KUKA KRL program: sample_robot_pick_place.src, sample_robot_pick_place.dat

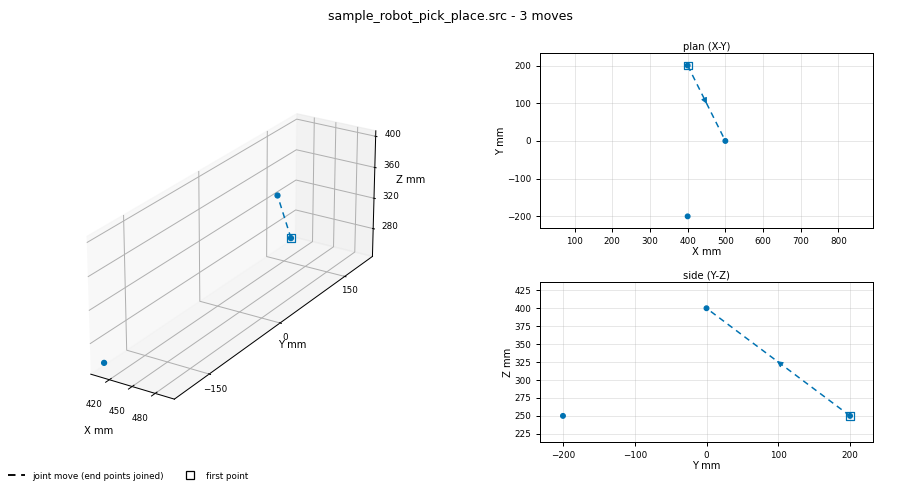
[picture p0: tool path of sample_robot_pick_place.src, 3 of 9 moves have a stored position in this frame; points joined in program order, loops and branches not executed]
--- sample_robot_pick_place.src ---
&ACCESS RVP
&REL 1
&PARAM TEMPLATE = C:\KRC\Roboter\Template\vorgabe
&PARAM EDITMASK = *

DEF sample_robot_pick_place()

; Sample KUKA robot program for pick and place operation
; This demonstrates typical KRL syntax and robot movements

; Variable declarations
DECL POS home_pos
DECL POS pick_pos
DECL POS place_pos
DECL INT counter
DECL BOOL gripper_state

; Initialize variables
counter = 0
gripper_state = FALSE
home_pos = {X 600.0, Y 0.0, Z 600.0, A 0.0, B 0.0, C 0.0}
pick_pos = {X 400.0, Y 200.0, Z 150.0, A 0.0, B 90.0, C 0.0}
place_pos = {X 400.0, Y -200.0, Z 150.0, A 0.0, B 90.0, C 0.0}

; Main program loop
FOR counter = 1 TO 5

  ; Move to home position
  PTP home_pos VEL=100 % DEFAULT

  ; Move to pick position
  PTP pick_pos VEL=50 % FINE

  ; Approach pick position
  LIN pick_pos VEL=10 % FINE

  ; Close gripper
  gripper_state = TRUE
  $OUT[1] = gripper_state
  WAIT SEC 0.5

  ; Lift part
  LIN {X 400.0, Y 200.0, Z 250.0, A 0.0, B 90.0, C 0.0} VEL=20 % FINE

  ; Move to place position (via intermediate point)
  PTP {X 500.0, Y 0.0, Z 400.0, A 0.0, B 45.0, C 0.0} VEL=75 % DEFAULT

  ; Approach place position
  PTP place_pos VEL=50 % FINE
  LIN place_pos VEL=10 % FINE

  ; Open gripper
  gripper_state = FALSE
  $OUT[1] = gripper_state
  WAIT SEC 0.5

  ; Retract
  LIN {X 400.0, Y -200.0, Z 250.0, A 0.0, B 90.0, C 0.0} VEL=20 % FINE

  ; Check safety conditions
  IF $IN[10] == TRUE THEN
    HALT
  ENDIF

ENDFOR

; Return to home
PTP home_pos VEL=100 % DEFAULT

END

--- sample_robot_pick_place.dat ---
&ACCESS RVP
&REL 1
&PARAM TEMPLATE = C:\KRC\Roboter\Template\vorgabe
&PARAM EDITMASK = *

DEFDAT sample_robot_pick_place

; Tool data for gripper
DECL FRAME TOOL_DATA[1] = {X 0.0, Y 0.0, Z 150.0, A 0.0, B 0.0, C 0.0}

; Base frame data
DECL FRAME BASE_DATA[1] = {X 0.0, Y 0.0, Z 0.0, A 0.0, B 0.0, C 0.0}

; Workpiece positions
DECL POS PICK_POINT[10]
DECL POS PLACE_POINT[10]

; Initialize pick points
PICK_POINT[1] = {X 400.0, Y 200.0, Z 150.0, A 0.0, B 90.0, C 0.0, S 2, T 35}
PICK_POINT[2] = {X 420.0, Y 200.0, Z 150.0, A 0.0, B 90.0, C 0.0, S 2, T 35}
PICK_POINT[3] = {X 440.0, Y 200.0, Z 150.0, A 0.0, B 90.0, C 0.0, S 2, T 35}

; Initialize place points
PLACE_POINT[1] = {X 400.0, Y -200.0, Z 150.0, A 0.0, B 90.0, C 0.0, S 2, T 35}
PLACE_POINT[2] = {X 420.0, Y -200.0, Z 150.0, A 0.0, B 90.0, C 0.0, S 2, T 35}
PLACE_POINT[3] = {X 440.0, Y -200.0, Z 150.0, A 0.0, B 90.0, C 0.0, S 2, T 35}

; Speed and zone data
DECL REAL VEL_FAST = 100.0
DECL REAL VEL_MEDIUM = 50.0
DECL REAL VEL_SLOW = 10.0

; Safety zone limits
DECL REAL X_MIN = -1000.0
DECL REAL X_MAX = 1000.0
DECL REAL Y_MIN = -1000.0
DECL REAL Y_MAX = 1000.0
DECL REAL Z_MIN = 0.0
DECL REAL Z_MAX = 2000.0

; Gripper configuration
DECL INT GRIPPER_OPEN_OUTPUT = 1
DECL INT GRIPPER_CLOSE_OUTPUT = 2
DECL INT PART_DETECT_INPUT = 10
DECL INT SAFETY_STOP_INPUT = 11

; Timer values
DECL REAL GRIPPER_DELAY = 0.5
DECL REAL SETTLE_TIME = 0.2

ENDDAT
